Yaskawa INFORM job: AAA.JBI

/JOB
//NAME AAA
//POS
///NPOS 4,0,0,0,0,0
///TOOL 1
///POSTYPE PULSE
///PULSE
C00000=0,-5294,-57573,0,56284,0
C00001=0,48804,15985,0,-18224,0
C00002=0,-5294,-57573,0,56284,0
C00003=0,48804,15985,0,-18224,0
//INST
///DATE 2022/11/22 15:01
///COMM Generated using RoboDK
///ATTR SC,RW
///GROUP1 RB2
NOP
'Using Motoman MA1440 Base (ta
'rgets wrt base):
'0.0,0.0,0.0,0.0,0.0,0.0
MOVJ C00000 VJ=5.0 PL=0
MOVJ C00001 VJ=5.0 PL=0
MOVJ C00002 VJ=5.0 PL=0
MOVJ C00003 VJ=5.0 PL=0
END
